TYPE State : BOOL; END_TYPE

(* stored: Version 1.1.0.1
   DUT State: Id {86a61754-313b-4526-8db1-641aa67db79c} *)
